// TwinCAT 3 PLC project rixs_optics
// Title: rix optics
// Company: SLAC
// ProjectVersion: 0.0.0
// ProgramVersion: 3.1.4022.7
// libraries:
//   LCLS General, * (SLAC)
//   lcls-twincat-motion, * (SLAC)
//   lcls-twincat-optics, * (SLAC)
//   PMPS, * (SLAC - LCLS)
//   Tc2_MC2, * (Beckhoff Automation GmbH)
//   Tc2_SerialCom, * (Beckhoff Automation GmbH)
//   Tc2_Standard, * (Beckhoff Automation GmbH)
//   Tc2_TcpIp, * (Beckhoff Automation GmbH)
//   Tc2_Utilities, * (Beckhoff Automation GmbH)
//   Tc3_Module, * (Beckhoff Automation GmbH)
// project tree:
//   GVLs/ GVL_DCCM_MONO.TcGVL, Main.TcGVL
//   Implicit Checks/ CheckBounds.TcPOU (not stored), CheckDivDInt.TcPOU (not stored), CheckDivLInt.TcPOU (not stored), CheckDivLReal.TcPOU (not stored), CheckDivReal.TcPOU (not stored), CheckLRangeSigned.TcPOU (not stored), CheckLRangeUnsigned.TcPOU (not stored), CheckPointer.TcPOU (not stored), CheckRangeSigned.TcPOU (not stored), CheckRangeUnsigned.TcPOU (not stored)
//   / PlcTask.TcTTO
//   POUs/ PRG_1_PlcTask.TcPOU, PRG_DCCM_MONO.TcPOU
// real-time tasks:
//   TASK PRG_1_PlcTask: cycle T#10ms, priority 20, ADS port 350
// motion (NC):
//   TASK NC-Task 1 SAF: cycle T#2ms, priority 4, ADS port 501
//   TASK NC-Task 1 SVB: cycle T#10ms, priority 8, ADS port 511
//   AXIS DCCM-th1-M1 (id 19)
//     Dynamic: Acceleration=8.99313, Deceleration=8.99313, Jerk=27.7544
//     Velo: SlowManual=1, FastManual=2, Maximum=3.1
//     TargetPosControl: Range=0.001
//     OtherSettings: AllowMotionCmdToSlave=true, PulseDistancePos=0.5, PulseDistanceNeg=0.5
//     encoder EncType=1
//       EncPara: ScaleFactorNumerator=1.2657e-07, Offset=-4.6852
//         SoftEndMinControl: Enable=true, Range=-3.7
//         SoftEndMaxControl: Enable=true, Range=3
//         Inc: RefSoftSyncMask=#x0000ffff
//     drive DrvType=24
//       DrvPara: Inverse=true
//         Analog: VeloReferenz=2, TorqueSetpointScale=10, ScaleFactorActTorque=0.1
//         TimeComp: TaskDelayCycles=1
//     controller CtrType=3
//       CtrPara: PriorControlFactor=1
//         PosDiffControl: Range=0.2
//         PID: PosKp=10, PosTv=0.2, DeadBandPosition=0.0001
//         Observer: BandWidth=20
//   AXIS DCCM-th2-M2 (id 20)
//     Dynamic: Acceleration=2.95205, Deceleration=2.95205, Jerk=8.98412
//     Velo: SlowManual=0.1, FastManual=0.3, Maximum=1
//     PositionAreaControl: Range=0.05
//     TargetPosControl: Range=0.0001
//     OtherSettings: AllowMotionCmdToSlave=true
//     encoder EncType=1
//       EncPara: ScaleFactorNumerator=1e-06, Offset=-10.712
//         SoftEndMinControl: Enable=true, Range=-4.15
//         SoftEndMaxControl: Enable=true, Range=3.15
//         Inc: RefSoftSyncMask=#x0000ffff
//     drive DrvType=24
//       DrvPara: Inverse=true
//         Analog: VeloReferenz=2, ScaleFactorActTorque=0.1
//         TimeComp: TaskDelayCycles=1
//     controller CtrType=3
//       CtrPara: PriorControlFactor=1
//         PosDiffControl: Range=0.15
//         PID: PosKp=7, PosTv=0.2
//         Observer: BandWidth=20
//   AXIS DCCM-tx-M3 (id 21)
//     Dynamic: Acceleration=0.424188, Deceleration=0.424188, Jerk=6.42628
//     Velo: SlowManual=0.3, FastManual=1, Maximum=2.8
//     PositionAreaControl: Range=0.2
//     TargetPosControl: Range=0.0005
//     OtherSettings: AllowMotionCmdToSlave=true, PulseDistancePos=1, PulseDistanceNeg=1
//     encoder EncType=1
//       EncPara: ScaleFactorNumerator=2.4267e-07, Offset=-1031.2195
//         SoftEndMinControl: Enable=true, Range=-4.82
//         SoftEndMaxControl: Enable=true, Range=6.22
//         Inc: RefSoftSyncMask=#x0000ffff
//     drive DrvType=24
//       Analog: VeloReferenz=2, ScaleFactorActTorque=0.1
//       TimeComp: TaskDelayCycles=1
//     controller CtrType=3
//       CtrPara: PriorControlFactor=1
//         PosDiffControl: Range=0.5
//         PID: PosKp=10, PosTv=0.2, DeadBandPosition=0.0001
//         Observer: BandWidth=20
//   AXIS DCCM-txd-M4 (id 22)
//     Dynamic: Acceleration=1.59597, Deceleration=1.59597, Jerk=4.61435
//     Velo: SlowManual=0.075, FastManual=0.2, Maximum=0.6
//     PositionAreaControl: Range=0.01
//     TargetPosControl: Range=0.0001
//     OtherSettings: AllowMotionCmdToSlave=true, PulseDistancePos=0.05, PulseDistanceNeg=0.05
//     encoder EncType=1
//       EncPara: ScaleFactorNumerator=1e-06, Offset=-19.5307
//         SoftEndMinControl: Enable=true, Range=0.02
//         SoftEndMaxControl: Enable=true, Range=8.65
//         Inc: RefSoftSyncMask=#x0000ffff
//     drive DrvType=24
//       DrvPara: Inverse=true
//         Analog: VeloReferenz=2, ScaleFactorActTorque=0.1
//         TimeComp: TaskDelayCycles=1
//     controller CtrType=3
//       CtrPara: PriorControlFactor=1
//         PosDiffControl: Range=0.15
//         PID: PosKp=4, PosTv=0.2, PosTd=1, DeadBandPosition=0.0001
//         Observer: BandWidth=20
//   AXIS DCCM-tyd-M5 (id 23)
//     Dynamic: Acceleration=4.26689, Deceleration=4.26689, Jerk=19.1646
//     Velo: SlowManual=0.5, FastManual=1, Maximum=2
//     PositionAreaControl: Range=0.05
//     TargetPosControl: Range=0.05
//     OtherSettings: AllowMotionCmdToSlave=true
//     encoder EncType=4
//       EncPara: ScaleFactorNumerator=1e-06, Offset=-17, MaxCount=#x0000ffff
//         SoftEndMinControl: Enable=true, Range=-0.59
//         SoftEndMaxControl: Enable=true, Range=41.6
//         Inc: RefMode=2, RefSoftSyncMask=#x0000ffff
//     drive DrvType=24
//       Analog: VeloReferenz=2, ScaleFactorActTorque=0.1
//       TimeComp: TaskDelayCycles=1
//     controller CtrType=3
//       CtrPara: PriorControlFactor=1
//         PosDiffControl: Range=1
//         PID: PosKp=15, PosTv=0.2, DeadBandPosition=0.01
//         Observer: BandWidth=20
//   AXIS DCCM-th1-M1_encoder (id 1)
//     OtherSettings: AllowMotionCmdToSlave=true
//     encoder EncType=29
//       EncPara: ScaleFactorNumerator=5, ScaleFactorDenominator=1000000, MaxCount=#xffffffff, MaxCountHighDWord=#x0000001f
//     drive DrvType=5
//       Analog: TorqueSetpointScale=10, ScaleFactorActTorque=0.1
//       TimeComp: TaskDelayCycles=1
//     controller CtrType=1
//       CtrPara: PriorControlFactor=1
//         Observer: BandWidth=20
//   AXIS DCCM-th2-M2_encoder (id 2)
//     OtherSettings: AllowMotionCmdToSlave=true
//     encoder EncType=29
//       EncPara: ScaleFactorNumerator=5, ScaleFactorDenominator=1000000, MaxCount=#xffffffff, MaxCountHighDWord=#x0000001f
//     drive DrvType=5
//       Analog: TorqueSetpointScale=10, ScaleFactorActTorque=0.1
//       TimeComp: TaskDelayCycles=1
//     controller CtrType=1
//       CtrPara: PriorControlFactor=1
//         Observer: BandWidth=20
//   AXIS DCCM-tx-M3_encoder (id 3)
//     OtherSettings: AllowMotionCmdToSlave=true
//     encoder EncType=29
//       EncPara: ScaleFactorNumerator=5, ScaleFactorDenominator=1000000, MaxCount=#xffffffff, MaxCountHighDWord=#x0000001f
//     drive DrvType=5
//       Analog: TorqueSetpointScale=10, ScaleFactorActTorque=0.1
//       TimeComp: TaskDelayCycles=1
//     controller CtrType=1
//       CtrPara: PriorControlFactor=1
//         Observer: BandWidth=20
//   AXIS DCCM-txd-M4_encoder (id 4)
//     OtherSettings: AllowMotionCmdToSlave=true
//     encoder EncType=29
//       EncPara: ScaleFactorNumerator=5, ScaleFactorDenominator=1000000, MaxCount=#xffffffff, MaxCountHighDWord=#x0000001f
//     drive DrvType=5
//       Analog: TorqueSetpointScale=10, ScaleFactorActTorque=0.1
//       TimeComp: TaskDelayCycles=1
//     controller CtrType=1
//       CtrPara: PriorControlFactor=1
//         Observer: BandWidth=20
//   AXIS DCCM-tyd-M5_encoder (id 5)
//     OtherSettings: AllowMotionCmdToSlave=true
//     encoder EncType=29
//       EncPara: ScaleFactorNumerator=5, ScaleFactorDenominator=1000000, MaxCount=#xffffffff, MaxCountHighDWord=#x0000001f
//     drive DrvType=5
//       Analog: TorqueSetpointScale=10, ScaleFactorActTorque=0.1
//       TimeComp: TaskDelayCycles=1
//     controller CtrType=1
//       CtrPara: PriorControlFactor=1
//         Observer: BandWidth=20
// I/O:
//   DEVICE Device 1 (EtherCAT) (disabled), AmsNetId 172.21.140.71.2.1
//     Term 1 (EK1200)
//   DEVICE Device 2 (EtherCAT), AmsNetId 0.0.0.0.3.1
//     EK1200_DCCM [EK1200-5000 EtherCAT Power supply (2A E-Bus)]
//       EL7047_DCCM_th1 [EL7047 1Ch. Stepper motor output stage (50V, 5A)]
//       EL7047_DCCM_th2 [EL7047 1Ch. Stepper motor output stage (50V, 5A)]
//       EL7047_DCCM_tx [EL7047 1Ch. Stepper motor output stage (50V, 5A)]
//       EL7047_DCCM_txd [EL7047 1Ch. Stepper motor output stage (50V, 5A)]
//       EL7047_DCCM_tyd [EL7047 1Ch. Stepper motor output stage (50V, 5A)]
//       EL5042_DCCM_th1_th2 [EL5042 2Ch. BiSS-C Encoder]
//       EL5042_DCCM_tx_txd [EL5042 2Ch. BiSS-C Encoder]
//       EL5042_DCCM_tyd [EL5042 2Ch. BiSS-C Encoder]
//       EL1008_DCCM_STO_DI [EL1008 8Ch. Dig. Input 24V, 3ms]
//       EL2008_DCCM_DO [EL2008 8Ch. Dig. Output 24V, 0.5A]
//       EL3062_DCCM_A1_C1 [EL3062 2Ch. Ana. Input 0-10V]
//       Term 13 (EL9011) [EL9011 End Terminal]
// variable links:
//   Axes/DCCM-th1-M1 <-> Device 2 (EtherCAT)/EK1200_DCCM/EL7047_DCCM_th1
//     Drive/Inputs/In/nState1 @bit 3 <-> STM Status/Status/Error
//     Drive/Inputs/In/nState1 @bit 7 <-> STM Status/Status/Motor stall
//     Drive/Inputs/In/nState1 @bit 5 <-> STM Status/Status/Moving negative
//     Drive/Inputs/In/nState1 @bit 4 <-> STM Status/Status/Moving positive
//     Drive/Inputs/In/nState1 @bit 1 <-> STM Status/Status/Ready
//     Drive/Inputs/In/nState1 <-> STM Status/Status/Ready to enable
//     Drive/Inputs/In/nState1 @bit 6 <-> STM Status/Status/Torque reduced
//     Drive/Inputs/In/nState1 @bit 2 <-> STM Status/Status/Warning
//     Drive/Inputs/In/nState2 @bit 3 <-> STM Status/Status/Digital input 1
//     Drive/Inputs/In/nState2 @bit 4 <-> STM Status/Status/Digital input 2
//     Drive/Inputs/In/nState2 @bit 5 <-> STM Status/Status/Sync error
//     Drive/Inputs/In/nState2 @bit 7 <-> STM Status/Status/TxPDO Toggle
//     Drive/Inputs/In/nState4 @bit 1 <-> WcState/InputToggle
//     Drive/Inputs/In/nState4 <-> WcState/WcState
//     Drive/Outputs/Out/nCtrl1 <-> STM Control/Control/Enable
//     Drive/Outputs/Out/nCtrl1 @bit 2 <-> STM Control/Control/Reduce torque
//     Drive/Outputs/Out/nCtrl1 @bit 1 <-> STM Control/Control/Reset
//     Drive/Outputs/Out/nCtrl2 @bit 3 <-> STM Control/Control/Digital output 1
//     Drive/Outputs/Out/nDataOut2[0] <-> STM Velocity/Velocity
//     Enc/Inputs/In/nDataIn1[0] <-> ENC Status compact/Counter value
//     Enc/Inputs/In/nDataIn2[0] <-> ENC Status compact/Latch value
//     Enc/Inputs/In/nState1 @bit 4 <-> ENC Status compact/Status/Counter overflow
//     Enc/Inputs/In/nState1 @bit 3 <-> ENC Status compact/Status/Counter underflow
//     Enc/Inputs/In/nState1 @bit 7 <-> ENC Status compact/Status/Extrapolation stall
//     Enc/Inputs/In/nState1 <-> ENC Status compact/Status/Latch C valid
//     Enc/Inputs/In/nState1 @bit 1 <-> ENC Status compact/Status/Latch extern valid
//     Enc/Inputs/In/nState1 @bit 2 <-> ENC Status compact/Status/Set counter done
//     Enc/Inputs/In/nState2 @bit 4 <-> ENC Status compact/Status/Status of extern latch
//     Enc/Inputs/In/nState2 <-> ENC Status compact/Status/Status of input A
//     Enc/Inputs/In/nState2 @bit 1 <-> ENC Status compact/Status/Status of input B
//     Enc/Inputs/In/nState2 @bit 2 <-> ENC Status compact/Status/Status of input C
//     Enc/Inputs/In/nState2 @bit 5 <-> ENC Status compact/Status/Sync error
//     Enc/Inputs/In/nState2 @bit 7 <-> ENC Status compact/Status/TxPDO Toggle
//     Enc/Inputs/In/nState4 @bit 1 <-> WcState/InputToggle
//     Enc/Inputs/In/nState4 <-> WcState/WcState
//     Enc/Outputs/Out/nCtrl1 <-> ENC Control compact/Control/Enable latch C
//     Enc/Outputs/Out/nCtrl1 @bit 3 <-> ENC Control compact/Control/Enable latch extern on negative edge
//     Enc/Outputs/Out/nCtrl1 @bit 1 <-> ENC Control compact/Control/Enable latch extern on positive edge
//     Enc/Outputs/Out/nCtrl1 @bit 2 <-> ENC Control compact/Control/Set counter
//     Enc/Outputs/Out/nDataOut1[0] <-> ENC Control compact/Set counter value
//   Axes/DCCM-th1-M1_encoder <-> Device 2 (EtherCAT)/EK1200_DCCM/EL5042_DCCM_th1_th2
//     Enc/Inputs/In/nComState @bit 1 <-> WcState/InputToggle
//     Enc/Inputs/In/nComState <-> WcState/WcState
//     Enc/Inputs/In/nDataIn1 <-> FB Inputs Channel 1/Position
//     Enc/Inputs/In/nState1 @bit 12 <-> FB Inputs Channel 1/Status/Diag
//     Enc/Inputs/In/nState1 @bit 1 <-> FB Inputs Channel 1/Status/Error
//     Enc/Inputs/In/nState1 @bit 14 <-> FB Inputs Channel 1/Status/Input cycle counter
//     Enc/Inputs/In/nState1 @bit 2 <-> FB Inputs Channel 1/Status/Ready
//     Enc/Inputs/In/nState1 @bit 13 <-> FB Inputs Channel 1/Status/TxPDO State
//     Enc/Inputs/In/nState1 <-> FB Inputs Channel 1/Status/Warning
//   Axes/DCCM-th2-M2 <-> Device 2 (EtherCAT)/EK1200_DCCM/EL7047_DCCM_th2
//     Drive/Inputs/In/nState1 @bit 3 <-> STM Status/Status/Error
//     Drive/Inputs/In/nState1 @bit 7 <-> STM Status/Status/Motor stall
//     Drive/Inputs/In/nState1 @bit 5 <-> STM Status/Status/Moving negative
//     Drive/Inputs/In/nState1 @bit 4 <-> STM Status/Status/Moving positive
//     Drive/Inputs/In/nState1 @bit 1 <-> STM Status/Status/Ready
//     Drive/Inputs/In/nState1 <-> STM Status/Status/Ready to enable
//     Drive/Inputs/In/nState1 @bit 6 <-> STM Status/Status/Torque reduced
//     Drive/Inputs/In/nState1 @bit 2 <-> STM Status/Status/Warning
//     Drive/Inputs/In/nState2 @bit 3 <-> STM Status/Status/Digital input 1
//     Drive/Inputs/In/nState2 @bit 4 <-> STM Status/Status/Digital input 2
//     Drive/Inputs/In/nState2 @bit 5 <-> STM Status/Status/Sync error
//     Drive/Inputs/In/nState2 @bit 7 <-> STM Status/Status/TxPDO Toggle
//     Drive/Inputs/In/nState4 @bit 1 <-> WcState/InputToggle
//     Drive/Inputs/In/nState4 <-> WcState/WcState
//     Drive/Outputs/Out/nCtrl1 <-> STM Control/Control/Enable
//     Drive/Outputs/Out/nCtrl1 @bit 2 <-> STM Control/Control/Reduce torque
//     Drive/Outputs/Out/nCtrl1 @bit 1 <-> STM Control/Control/Reset
//     Drive/Outputs/Out/nCtrl2 @bit 3 <-> STM Control/Control/Digital output 1
//     Drive/Outputs/Out/nDataOut2[0] <-> STM Velocity/Velocity
//   Axes/DCCM-th2-M2_encoder <-> Device 2 (EtherCAT)/EK1200_DCCM/EL5042_DCCM_th1_th2
//     Enc/Inputs/In/nComState @bit 1 <-> WcState/InputToggle
//     Enc/Inputs/In/nComState <-> WcState/WcState
//     Enc/Inputs/In/nDataIn1 <-> FB Inputs Channel 2/Position
//     Enc/Inputs/In/nState1 @bit 12 <-> FB Inputs Channel 2/Status/Diag
//     Enc/Inputs/In/nState1 @bit 1 <-> FB Inputs Channel 2/Status/Error
//     Enc/Inputs/In/nState1 @bit 14 <-> FB Inputs Channel 2/Status/Input cycle counter
//     Enc/Inputs/In/nState1 @bit 2 <-> FB Inputs Channel 2/Status/Ready
//     Enc/Inputs/In/nState1 @bit 13 <-> FB Inputs Channel 2/Status/TxPDO State
//     Enc/Inputs/In/nState1 <-> FB Inputs Channel 2/Status/Warning
//   Axes/DCCM-tx-M3 <-> Device 2 (EtherCAT)/EK1200_DCCM/EL7047_DCCM_tx
//     Drive/Inputs/In/nState1 @bit 3 <-> STM Status/Status/Error
//     Drive/Inputs/In/nState1 @bit 7 <-> STM Status/Status/Motor stall
//     Drive/Inputs/In/nState1 @bit 5 <-> STM Status/Status/Moving negative
//     Drive/Inputs/In/nState1 @bit 4 <-> STM Status/Status/Moving positive
//     Drive/Inputs/In/nState1 @bit 1 <-> STM Status/Status/Ready
//     Drive/Inputs/In/nState1 <-> STM Status/Status/Ready to enable
//     Drive/Inputs/In/nState1 @bit 6 <-> STM Status/Status/Torque reduced
//     Drive/Inputs/In/nState1 @bit 2 <-> STM Status/Status/Warning
//     Drive/Inputs/In/nState2 @bit 3 <-> STM Status/Status/Digital input 1
//     Drive/Inputs/In/nState2 @bit 4 <-> STM Status/Status/Digital input 2
//     Drive/Inputs/In/nState2 @bit 5 <-> STM Status/Status/Sync error
//     Drive/Inputs/In/nState2 @bit 7 <-> STM Status/Status/TxPDO Toggle
//     Drive/Inputs/In/nState4 @bit 1 <-> WcState/InputToggle
//     Drive/Inputs/In/nState4 <-> WcState/WcState
//     Drive/Outputs/Out/nCtrl1 <-> STM Control/Control/Enable
//     Drive/Outputs/Out/nCtrl1 @bit 2 <-> STM Control/Control/Reduce torque
//     Drive/Outputs/Out/nCtrl1 @bit 1 <-> STM Control/Control/Reset
//     Drive/Outputs/Out/nCtrl2 @bit 3 <-> STM Control/Control/Digital output 1
//     Drive/Outputs/Out/nDataOut2[0] <-> STM Velocity/Velocity
//   Axes/DCCM-tx-M3_encoder <-> Device 2 (EtherCAT)/EK1200_DCCM/EL5042_DCCM_tx_txd
//     Enc/Inputs/In/nComState @bit 1 <-> WcState/InputToggle
//     Enc/Inputs/In/nComState <-> WcState/WcState
//     Enc/Inputs/In/nDataIn1 <-> FB Inputs Channel 1/Position
//     Enc/Inputs/In/nState1 @bit 12 <-> FB Inputs Channel 1/Status/Diag
//     Enc/Inputs/In/nState1 @bit 1 <-> FB Inputs Channel 1/Status/Error
//     Enc/Inputs/In/nState1 @bit 14 <-> FB Inputs Channel 1/Status/Input cycle counter
//     Enc/Inputs/In/nState1 @bit 2 <-> FB Inputs Channel 1/Status/Ready
//     Enc/Inputs/In/nState1 @bit 13 <-> FB Inputs Channel 1/Status/TxPDO State
//     Enc/Inputs/In/nState1 <-> FB Inputs Channel 1/Status/Warning
//   Axes/DCCM-txd-M4 <-> Device 2 (EtherCAT)/EK1200_DCCM/EL7047_DCCM_txd
//     Drive/Inputs/In/nState1 @bit 3 <-> STM Status/Status/Error
//     Drive/Inputs/In/nState1 @bit 7 <-> STM Status/Status/Motor stall
//     Drive/Inputs/In/nState1 @bit 5 <-> STM Status/Status/Moving negative
//     Drive/Inputs/In/nState1 @bit 4 <-> STM Status/Status/Moving positive
//     Drive/Inputs/In/nState1 @bit 1 <-> STM Status/Status/Ready
//     Drive/Inputs/In/nState1 <-> STM Status/Status/Ready to enable
//     Drive/Inputs/In/nState1 @bit 6 <-> STM Status/Status/Torque reduced
//     Drive/Inputs/In/nState1 @bit 2 <-> STM Status/Status/Warning
//     Drive/Inputs/In/nState2 @bit 3 <-> STM Status/Status/Digital input 1
//     Drive/Inputs/In/nState2 @bit 4 <-> STM Status/Status/Digital input 2
//     Drive/Inputs/In/nState2 @bit 5 <-> STM Status/Status/Sync error
//     Drive/Inputs/In/nState2 @bit 7 <-> STM Status/Status/TxPDO Toggle
//     Drive/Inputs/In/nState4 @bit 1 <-> WcState/InputToggle
//     Drive/Inputs/In/nState4 <-> WcState/WcState
//     Drive/Outputs/Out/nCtrl1 <-> STM Control/Control/Enable
//     Drive/Outputs/Out/nCtrl1 @bit 2 <-> STM Control/Control/Reduce torque
//     Drive/Outputs/Out/nCtrl1 @bit 1 <-> STM Control/Control/Reset
//     Drive/Outputs/Out/nCtrl2 @bit 3 <-> STM Control/Control/Digital output 1
//     Drive/Outputs/Out/nDataOut2[0] <-> STM Velocity/Velocity
//   Axes/DCCM-txd-M4_encoder <-> Device 2 (EtherCAT)/EK1200_DCCM/EL5042_DCCM_tx_txd
//     Enc/Inputs/In/nComState @bit 1 <-> WcState/InputToggle
//     Enc/Inputs/In/nComState <-> WcState/WcState
//     Enc/Inputs/In/nDataIn1 <-> FB Inputs Channel 2/Position
//     Enc/Inputs/In/nState1 @bit 12 <-> FB Inputs Channel 2/Status/Diag
//     Enc/Inputs/In/nState1 @bit 1 <-> FB Inputs Channel 2/Status/Error
//     Enc/Inputs/In/nState1 @bit 14 <-> FB Inputs Channel 2/Status/Input cycle counter
//     Enc/Inputs/In/nState1 @bit 2 <-> FB Inputs Channel 2/Status/Ready
//     Enc/Inputs/In/nState1 @bit 13 <-> FB Inputs Channel 2/Status/TxPDO State
//     Enc/Inputs/In/nState1 <-> FB Inputs Channel 2/Status/Warning
//   Axes/DCCM-tyd-M5 <-> Device 2 (EtherCAT)/EK1200_DCCM/EL7047_DCCM_tyd
//     Drive/Inputs/In/nState1 @bit 3 <-> STM Status/Status/Error
//     Drive/Inputs/In/nState1 @bit 7 <-> STM Status/Status/Motor stall
//     Drive/Inputs/In/nState1 @bit 5 <-> STM Status/Status/Moving negative
//     Drive/Inputs/In/nState1 @bit 4 <-> STM Status/Status/Moving positive
//     Drive/Inputs/In/nState1 @bit 1 <-> STM Status/Status/Ready
//     Drive/Inputs/In/nState1 <-> STM Status/Status/Ready to enable
//     Drive/Inputs/In/nState1 @bit 6 <-> STM Status/Status/Torque reduced
//     Drive/Inputs/In/nState1 @bit 2 <-> STM Status/Status/Warning
//     Drive/Inputs/In/nState2 @bit 3 <-> STM Status/Status/Digital input 1
//     Drive/Inputs/In/nState2 @bit 4 <-> STM Status/Status/Digital input 2
//     Drive/Inputs/In/nState2 @bit 5 <-> STM Status/Status/Sync error
//     Drive/Inputs/In/nState2 @bit 7 <-> STM Status/Status/TxPDO Toggle
//     Drive/Inputs/In/nState4 @bit 1 <-> WcState/InputToggle
//     Drive/Inputs/In/nState4 <-> WcState/WcState
//     Drive/Outputs/Out/nCtrl1 <-> STM Control/Control/Enable
//     Drive/Outputs/Out/nCtrl1 @bit 2 <-> STM Control/Control/Reduce torque
//     Drive/Outputs/Out/nCtrl1 @bit 1 <-> STM Control/Control/Reset
//     Drive/Outputs/Out/nCtrl2 @bit 3 <-> STM Control/Control/Digital output 1
//     Drive/Outputs/Out/nDataOut2[0] <-> STM Velocity/Velocity
//     Enc/Inputs/In/nDataIn1[0] <-> ENC Status compact/Counter value
//     Enc/Inputs/In/nDataIn2[0] <-> ENC Status compact/Latch value
//     Enc/Inputs/In/nState1 @bit 4 <-> ENC Status compact/Status/Counter overflow
//     Enc/Inputs/In/nState1 @bit 3 <-> ENC Status compact/Status/Counter underflow
//     Enc/Inputs/In/nState1 @bit 7 <-> ENC Status compact/Status/Extrapolation stall
//     Enc/Inputs/In/nState1 <-> ENC Status compact/Status/Latch C valid
//     Enc/Inputs/In/nState1 @bit 1 <-> ENC Status compact/Status/Latch extern valid
//     Enc/Inputs/In/nState1 @bit 2 <-> ENC Status compact/Status/Set counter done
//     Enc/Inputs/In/nState2 @bit 4 <-> ENC Status compact/Status/Status of extern latch
//     Enc/Inputs/In/nState2 <-> ENC Status compact/Status/Status of input A
//     Enc/Inputs/In/nState2 @bit 1 <-> ENC Status compact/Status/Status of input B
//     Enc/Inputs/In/nState2 @bit 2 <-> ENC Status compact/Status/Status of input C
//     Enc/Inputs/In/nState2 @bit 5 <-> ENC Status compact/Status/Sync error
//     Enc/Inputs/In/nState2 @bit 7 <-> ENC Status compact/Status/TxPDO Toggle
//     Enc/Inputs/In/nState4 @bit 1 <-> WcState/InputToggle
//     Enc/Inputs/In/nState4 <-> WcState/WcState
//     Enc/Outputs/Out/nCtrl1 <-> ENC Control compact/Control/Enable latch C
//     Enc/Outputs/Out/nCtrl1 @bit 3 <-> ENC Control compact/Control/Enable latch extern on negative edge
//     Enc/Outputs/Out/nCtrl1 @bit 1 <-> ENC Control compact/Control/Enable latch extern on positive edge
//     Enc/Outputs/Out/nCtrl1 @bit 2 <-> ENC Control compact/Control/Set counter
//     Enc/Outputs/Out/nDataOut1[0] <-> ENC Control compact/Set counter value
//   Axes/DCCM-tyd-M5_encoder <-> Device 2 (EtherCAT)/EK1200_DCCM/EL5042_DCCM_tyd
//     Enc/Inputs/In/nComState @bit 1 <-> WcState/InputToggle
//     Enc/Inputs/In/nComState <-> WcState/WcState
//     Enc/Inputs/In/nDataIn1 <-> FB Inputs Channel 1/Position
//     Enc/Inputs/In/nState1 @bit 12 <-> FB Inputs Channel 1/Status/Diag
//     Enc/Inputs/In/nState1 @bit 1 <-> FB Inputs Channel 1/Status/Error
//     Enc/Inputs/In/nState1 @bit 14 <-> FB Inputs Channel 1/Status/Input cycle counter
//     Enc/Inputs/In/nState1 @bit 2 <-> FB Inputs Channel 1/Status/Ready
//     Enc/Inputs/In/nState1 @bit 13 <-> FB Inputs Channel 1/Status/TxPDO State
//     Enc/Inputs/In/nState1 <-> FB Inputs Channel 1/Status/Warning
//   rixs_optics Instance <-> Device 2 (EtherCAT)/EK1200_DCCM/EL1008_DCCM_STO_DI
//     PlcTask Outputs/PRG_DCCM_MONO.bDI7 <-> Channel 8/Input
//     PlcTask Outputs/PRG_DCCM_MONO.bSTO <-> Channel 7/Input
//     PlcTask Outputs/PRG_DCCM_MONO.bTH1_NOTL <-> Channel 2/Input
//     PlcTask Outputs/PRG_DCCM_MONO.bTH2_NOTL <-> Channel 4/Input
//     PlcTask Outputs/PRG_DCCM_MONO.bTH1_POTL <-> Channel 1/Input
//     PlcTask Outputs/PRG_DCCM_MONO.bTH2_POTL <-> Channel 3/Input
//     PlcTask Outputs/PRG_DCCM_MONO.bTX_NOTL <-> Channel 6/Input
//     PlcTask Outputs/PRG_DCCM_MONO.bTX_POTL <-> Channel 5/Input
//   rixs_optics Instance <-> Device 2 (EtherCAT)/EK1200_DCCM/EL2008_DCCM_DO
//     PlcTask Outputs/PRG_DCCM_MONO.bFanOn <-> Channel 8/Output
//   rixs_optics Instance <-> Device 2 (EtherCAT)/EK1200_DCCM/EL7047_DCCM_th1
//     PlcTask Inputs/Main.M1.bLimitBackwardEnable <-> STM Status/Status/Digital input 2
//     PlcTask Inputs/Main.M1.bLimitForwardEnable <-> STM Status/Status/Digital input 1
//   rixs_optics Instance <-> Device 2 (EtherCAT)/EK1200_DCCM/EL7047_DCCM_th2
//     PlcTask Inputs/Main.M2.bLimitBackwardEnable <-> STM Status/Status/Digital input 2
//     PlcTask Inputs/Main.M2.bLimitForwardEnable <-> STM Status/Status/Digital input 1
//   rixs_optics Instance <-> Device 2 (EtherCAT)/EK1200_DCCM/EL7047_DCCM_tx
//     PlcTask Inputs/Main.M3.bLimitBackwardEnable <-> STM Status/Status/Digital input 2
//     PlcTask Inputs/Main.M3.bLimitForwardEnable <-> STM Status/Status/Digital input 1
//   rixs_optics Instance <-> Device 2 (EtherCAT)/EK1200_DCCM/EL7047_DCCM_txd
//     PlcTask Inputs/Main.M4.bLimitBackwardEnable <-> STM Status/Status/Digital input 2
//     PlcTask Inputs/Main.M4.bLimitForwardEnable <-> STM Status/Status/Digital input 1
//   rixs_optics Instance <-> NC-Task 1 SAF/Axes/DCCM-th1-M1
//     PlcTask Inputs/Main.M1.Axis.NcToPlc <-> Outputs/ToPlc
//     PlcTask Outputs/Main.M1.Axis.PlcToNc <-> Inputs/FromPlc
//   rixs_optics Instance <-> NC-Task 1 SAF/Axes/DCCM-th2-M2
//     PlcTask Inputs/Main.M2.Axis.NcToPlc <-> Outputs/ToPlc
//     PlcTask Outputs/Main.M2.Axis.PlcToNc <-> Inputs/FromPlc
//   rixs_optics Instance <-> NC-Task 1 SAF/Axes/DCCM-tx-M3
//     PlcTask Inputs/Main.M3.Axis.NcToPlc <-> Outputs/ToPlc
//     PlcTask Outputs/Main.M3.Axis.PlcToNc <-> Inputs/FromPlc
//   rixs_optics Instance <-> NC-Task 1 SAF/Axes/DCCM-txd-M4
//     PlcTask Inputs/Main.M4.Axis.NcToPlc <-> Outputs/ToPlc
//     PlcTask Outputs/Main.M4.Axis.PlcToNc <-> Inputs/FromPlc
//   rixs_optics Instance <-> NC-Task 1 SAF/Axes/DCCM-tyd-M5
//     PlcTask Inputs/Main.M5.Axis.NcToPlc <-> Outputs/ToPlc
//     PlcTask Outputs/Main.M5.Axis.PlcToNc <-> Inputs/FromPlc

CONFIGURATION rixs_optics
    RESOURCE PLC ON TwinCAT3
        TASK PlcTask(INTERVAL := T#10ms, PRIORITY := 20);
        PROGRAM PRG_1_PlcTask WITH PlcTask : PRG_1_PlcTask;
    END_RESOURCE
END_CONFIGURATION

// ---- GVLs/GVL_DCCM_MONO.TcGVL
{attribute 'qualified_only'}
VAR_GLOBAL CONSTANT
    // Encoder reference values in counts = nm
    // Put encoder reference values for nominal 0 here
    nM2K2X_ENC_REF : ULINT := 6077000; //these numbers
    nM2K2Y_ENC_REF : ULINT := 5975460; //are
    nM2K2rX_ENC_REF : ULINT := 50412360;//real
END_VAR

// ---- GVLs/Main.TcGVL
VAR_GLOBAL
(*
    Only includes motor definitions for the IOC
    These are hard-coded to be Main.M#,
    but are very convenient to store in a GVL,
    hence the confusing namespace here

    This should be refactored once the IOC
    supports arbitrary ads paths for motors
*)
    (*DCCM Mono*)
    // Motors
	                                               
    {attribute 'TcLinkTo' := '.bLimitForwardEnable:=TIID^Device 2 (EtherCAT)^EK1200_DCCM^EL7047_DCCM_th1^STM Status^Status^Digital input 1;
                              .bLimitBackwardEnable:=TIID^Device 2 (EtherCAT)^EK1200_DCCM^EL7047_DCCM_th1^STM Status^Status^Digital input 2;'}
    {attribute 'pytmc' := '
        pv: DCCM:SWITCH:MMS:TH1
    '}
    M1 : DUT_MotionStage := (fVelocity:=100.0, nEnableMode:=ENUM_StageEnableMode.ALWAYS, bPowerSelf:=TRUE); // DCCM th1
    fbMotionStage_m1 : FB_MotionStage;

    {attribute 'TcLinkTo' := '.bLimitForwardEnable:=TIID^Device 2 (EtherCAT)^EK1200_DCCM^EL7047_DCCM_th2^STM Status^Status^Digital input 1;
                              .bLimitBackwardEnable:=TIID^Device 2 (EtherCAT)^EK1200_DCCM^EL7047_DCCM_th2^STM Status^Status^Digital input 2;'}
    {attribute 'pytmc' := '
        pv: DCCM:SWITCH:MMS:TH2
    '}
    M2 : DUT_MotionStage := (fVelocity:=100.0, nEnableMode:=ENUM_StageEnableMode.ALWAYS, bPowerSelf:=TRUE); // DCCM th2
    fbMotionStage_m2 : FB_MotionStage;

	{attribute 'TcLinkTo' := '.bLimitForwardEnable:=TIID^Device 2 (EtherCAT)^EK1200_DCCM^EL7047_DCCM_tx^STM Status^Status^Digital input 1;
                              .bLimitBackwardEnable:=TIID^Device 2 (EtherCAT)^EK1200_DCCM^EL7047_DCCM_tx^STM Status^Status^Digital input 2;'}
    {attribute 'pytmc' := '
        pv: DCCM:SWITCH:MMS:TX
    '}
    M3 : DUT_MotionStage := (fVelocity:=150.0, nEnableMode:=ENUM_StageEnableMode.ALWAYS, bPowerSelf:=TRUE); // DCCM tx
    fbMotionStage_m3 : FB_MotionStage;

    {attribute 'TcLinkTo' := '.bLimitForwardEnable:=TIID^Device 2 (EtherCAT)^EK1200_DCCM^EL7047_DCCM_txd^STM Status^Status^Digital input 1;
                              .bLimitBackwardEnable:=TIID^Device 2 (EtherCAT)^EK1200_DCCM^EL7047_DCCM_txd^STM Status^Status^Digital input 2;'}
    {attribute 'pytmc' := '
        pv: DCCM:SWITCH:MMS:TXD
    '}
    M4 : DUT_MotionStage := (fVelocity:=150.0, nEnableMode:=ENUM_StageEnableMode.ALWAYS, bPowerSelf:=TRUE); // DCCM txd
    fbMotionStage_m4 : FB_MotionStage;

    {attribute 'TcLinkTo' := '.bLimitForwardEnable:=TIID^Device 2 (EtherCAT)^EK1200_DCCM^EL7047_DCCM_txy^STM Status^Status^Digital input 1;
                              .bLimitBackwardEnable:=TIID^Device 2 (EtherCAT)^EK1200_DCCM^EL7047_DCCM_txy^STM Status^Status^Digital input 2;'}
    {attribute 'pytmc' := '
        pv: DCCM:SWITCH:MMS:txy
    '}
    M5 : DUT_MotionStage := (fVelocity:=30.0, nEnableMode:=ENUM_StageEnableMode.DURING_MOTION, bPowerSelf:=TRUE); // DCCM txy
	fbMotionStage_m5 : FB_MotionStage;	
END_VAR

// ---- POUs/PRG_1_PlcTask.TcPOU
PROGRAM PRG_1_PlcTask
VAR
//fbLogHandler: FB_LogHandler;
	// PRG_DCCM_MONO: INT;
END_VAR

PRG_DCCM_MONO();
//fbLogHandler();

END_PROGRAM

// ---- POUs/PRG_DCCM_MONO.TcPOU
PROGRAM PRG_DCCM_MONO
VAR
//    FFO    :    FB_FastFault :=(
//        i_DevName := 'DCCM-MONO',
//        i_Desc := 'Fault occurs when device is in an usafe state',
//        i_TypeCode := 16#E50);




    {attribute 'pytmc' := '
        pv: DCCM:MONO:FAN:PWR
        field: ZNAM OFF ;
        field: ONAM ON ;
    '}
     {attribute 'TcLinkTo' := 'TIID^Device 2 (EtherCAT)^EK1200_DCCM^EL2008_DCCM_DO^Channel 8^Output'}
    bFanOn AT %Q*:BOOL;
	

	
	{attribute 'pytmc' := '
        pv: DCCM:MONO:th1:POTL
        field: ZNAM OFF ;
        field: ONAM ON ;
    '}
	{attribute 'TcLinkTo' := 'TIID^Device 2 (EtherCAT)^EK1200_DCCM^EL1008_DCCM_STO_DI^Channel 1^Input'}
	bTH1_POTL AT %Q*:BOOL;
	
		{attribute 'pytmc' := '
        pv: DCCM:MONO:th1:NOTL
        field: ZNAM OFF ;
        field: ONAM ON ;
    '}
	{attribute 'TcLinkTo' := 'TIID^Device 2 (EtherCAT)^EK1200_DCCM^EL1008_DCCM_STO_DI^Channel 2^Input'}
	bTH1_NOTL AT %Q*:BOOL;
	
	{attribute 'pytmc' := '
        pv: DCCM:MONO:th2:POTL
        field: ZNAM OFF ;
        field: ONAM ON ;
    '}
	{attribute 'TcLinkTo' := 'TIID^Device 2 (EtherCAT)^EK1200_DCCM^EL1008_DCCM_STO_DI^Channel 3^Input'}
	bTH2_POTL AT %Q*:BOOL;
	
		{attribute 'pytmc' := '
        pv: DCCM:MONO:th2:NOTL
        field: ZNAM OFF ;
        field: ONAM ON ;
    '}
	{attribute 'TcLinkTo' := 'TIID^Device 2 (EtherCAT)^EK1200_DCCM^EL1008_DCCM_STO_DI^Channel 4^Input'}
	bTH2_NOTL AT %Q*:BOOL;
	
		{attribute 'pytmc' := '
        pv: DCCM:MONO:tx:POTL
        field: ZNAM OFF ;
        field: ONAM ON ;
    '}
	{attribute 'TcLinkTo' := 'TIID^Device 2 (EtherCAT)^EK1200_DCCM^EL1008_DCCM_STO_DI^Channel 5^Input'}
	bTX_POTL AT %Q*:BOOL;
	
		{attribute 'pytmc' := '
        pv: DCCM:MONO:tx:NOTL
        field: ZNAM OFF ;
        field: ONAM ON ;
    '}
	{attribute 'TcLinkTo' := 'TIID^Device 2 (EtherCAT)^EK1200_DCCM^EL1008_DCCM_STO_DI^Channel 6^Input'}
	bTX_NOTL AT %Q*:BOOL;
	
	
	{attribute 'pytmc' := '
        pv: DCCM:MONO:STO
        field: ZNAM OFF ;
        field: ONAM ON ;
    '}
	{attribute 'TcLinkTo' := 'TIID^Device 2 (EtherCAT)^EK1200_DCCM^EL1008_DCCM_STO_DI^Channel 7^Input'}
	bSTO AT %Q*:BOOL;

	{attribute 'pytmc' := '
        pv: DCCM:MONO:DI7
        field: ZNAM OFF ;
        field: ONAM ON ;
    '}
	{attribute 'TcLinkTo' := 'TIID^Device 2 (EtherCAT)^EK1200_DCCM^EL1008_DCCM_STO_DI^Channel 8^Input'}
	bDI7 AT %Q*:BOOL;
	
	{attribute 'pytmc' := '
        pv: DCCM:MONO:A1
    '}
	{attribute 'TcLinkTo' :=TIID^Device 2 (EtherCAT)^EK1200_DCCM^EL3062_DCCM_A1_C1^AI Standard Channel 1^Value'}
	wA1 AT %I*:INT;
	
	{attribute 'pytmc' := '
        pv: DCCM:MONO:C1
    '}
	{attribute 'TcLinkTo' :=TIID^Device 2 (EtherCAT)^EK1200_DCCM^EL3062_DCCM_A1_C1^AI Standard Channel 2^Value'}
	wC1 AT %I*:INT;

	
    bInit : BOOL:=TRUE;

     (*Motion Parameters*)
    fSmallDelta: LREAL := 0.01;
    fBigDelta: LREAL := 10;
    fMaxVelocity: LREAL := 0.5;
    fHighAccel: LREAL := 0.8;
    fLowAccel: LREAL := 0.1;

END_VAR

//  init the motion stages parameters
IF ( bInit) THEN
    bInit := FALSE;
//    FFO.i_DevName := 'DCCM-MONO';
    //Bragg 1
    
	Main.M1.bEnable:=TRUE;
    Main.M1.bPowerSelf :=TRUE;
    Main.M1.nBrakeMode := ENUM_StageBrakeMode.NO_BRAKE;
    Main.M1.nEnableMode := ENUM_StageEnableMode.DURING_MOTION;
   //Bragg 2
    
    Main.M2.bPowerSelf :=TRUE;
    Main.M2.nBrakeMode := ENUM_StageBrakeMode.NO_BRAKE;
    Main.M2.nEnableMode := ENUM_StageEnableMode.DURING_MOTION;
    //TX
    
    Main.M3.bPowerSelf :=TRUE;
    Main.M3.nBrakeMode := ENUM_StageBrakeMode.NO_BRAKE;
    Main.M3.nEnableMode := ENUM_StageEnableMode.DURING_MOTION;
    //TXD
    
    Main.M4.bPowerSelf :=TRUE;
    Main.M4.nBrakeMode := ENUM_StageBrakeMode.NO_BRAKE;
    Main.M4.nEnableMode := ENUM_StageEnableMode.DURING_MOTION;
    //TYD
    
    Main.M5.bPowerSelf :=TRUE;
    Main.M5.nBrakeMode := ENUM_StageBrakeMode.NO_BRAKE;
    Main.M5.nEnableMode := ENUM_StageEnableMode.DURING_MOTION;

    //Turn on Fan by default
    bFanOn := TRUE;
END_IF

 	fbMotionStage_m1  (stMotionStage:=M1);
	fbMotionStage_m2  (stMotionStage:=M2);
	fbMotionStage_m3  (stMotionStage:=M3);
	fbMotionStage_m4  (stMotionStage:=M4);
	fbMotionStage_m5  (stMotionStage:=M5);
	
	Main.M1.bHardwareEnable := bSTO AND bTH1_POTL AND bTH1_NOTL;
	Main.M2.bHardwareEnable := bSTO AND bTH2_POTL AND bTH2_NOTL;
	Main.M3.bHardwareEnable := bSTO AND bTX_POTL AND bTX_NOTL;

END_PROGRAM
